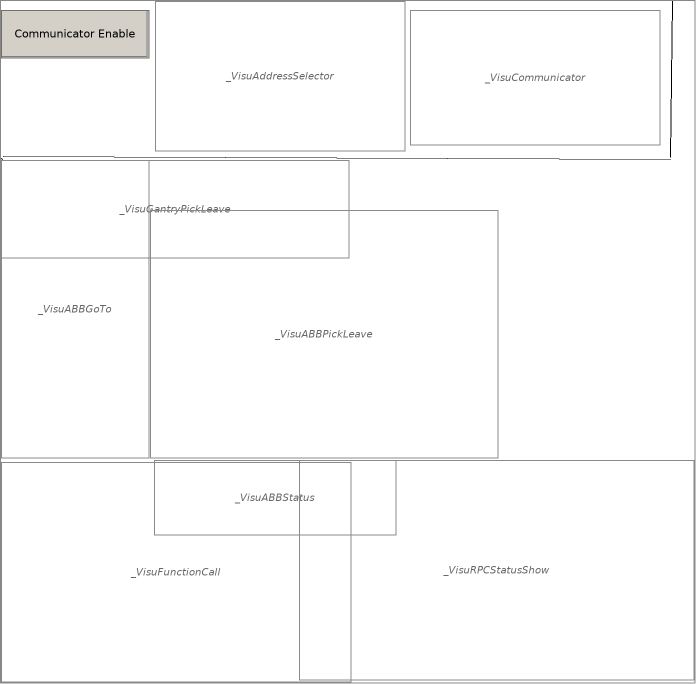
VISUALIZATION _TryOut  // 696x684
    Frame (1,160 148x298), invisible if: not ComGVL._fbTryOutShowABB
        shows _VisuABBGoTo()
    Button (1,10 148x48), "Communicator Enable"
    Frame (155,1 250x150), invisible if: ComGVL._mxTryOutEnable
        shows _VisuAddressSelector()
    Frame (1,160 348x98), invisible if: NOT ComGVL._fbTryOutShowGantry
        shows _VisuGantryPickLeave()
    Frame (150,210 348x248), invisible if: NOT ComGVL._fbTryOutShowABB
        shows _VisuABBPickLeave()
    Frame (154,460 242x75)
        shows _VisuABBStatus()
    Frame (1,462 350x220)
        shows _VisuFunctionCall()
    Frame (410,10 250x135)
        shows _VisuCommunicator()
    Line (1,158) (2,159)
    Line (3,156) (670,159)
    Line (672,1) (670,157)
    Frame (299,460 395x220)
        shows _VisuRPCStatusShow()
END_VISUALIZATION

(* stored: Version 1.1.0.1, ProductVersion 3.1.4024.2
   Visu _TryOut: Id {05910b5d-6908-4604-97d7-628369663da5} *)
